FUNCTION_BLOCK FB_InternalPowerSupply implements itf_standardFB

VAR
	IO									: FB_InternalPowerSupply_IO;
	UPS									: FB_UPS;
	InternalPowerDemand					: ST_InternalPowerSupply_PowerDemand;
	b_EMStopActive 						: BOOL := FALSE;
	b_killUPS							: BOOL := FALSE;	
	b_HVDCAllowed						: BOOL;
	
	rtrig_CEEConnected					:	r_trig;
	LowBatShutdownTimer					:	TON;
	
	UPSChargeMode	:	bool;
END_VAR

VAR_IN_OUT CONSTANT
	st_params							: 	ST_InternalPowerSupply_Params;
END_VAR

VAR_INPUT
	st_CoolingDemandSupply				: ST_InternalPowerSupply_PowerDemand;
	st_PowerstackDemandSupply			: ST_InternalPowerSupply_PowerDemand;
	st_ACDCChargerDemandSupply			: ST_InternalPowerSupply_PowerDemand;
	st_DCBusDemandSupply				: ST_InternalPowerSupply_PowerDemand;
	
	b_BusbarACAvailable					: BOOL	:=	FALSE;
	e_BMSPowerstate						: eHVDC_Powerstatus;
	b_ConditioningOnBatteryAllowed		:	BOOL;
END_VAR

VAR_OUTPUT
	Get									: ST_InternalPowerSupply_Get;
	b_HVDC_Enable						: BOOL;
	b_PowerStackACRequired				: BOOL;
END_VAR


var
	b_ACPSU_OK				at %i* :	Bool;
	b_DCPSU_OK				at %i* :	Bool;
	b_CEEInputAvailable		AT %i* : 	Bool;
	b_enableHVDCPSU			AT %Q* :	Bool;
END_VAR

// call functions
UPS(b_24v_available := get.b_24VdcAvailable, st_params := st_params);
	get.UPS REF= UPS.Get;

ACPowerControl(st_params:=st_params, get:=get);
DCPowerControl(st_params:=st_params, b_UPSDemand24VDC := ups.b_UPSDemand24VDC,  get:= get);
HVDCPowerControl(enable := b_HVDCAllowed);

//if ups battery low warning occurs and no 24V is available, charging request failed and the system shuts down.
//If the system is connected to a source (HVDC, CEE, powerlock or internal AC), this is skipped.
//In that case, LowBatteryError will trip a system shutdown
LowBatShutdownTimer(in := UPS.Get.Events.b_BatteryLowWarning AND NOT get.b_24VdcAvailable, PT := st_params.LowBatteryShutdownTimer);
IF LowBatShutdownTimer.Q THEN
	SystemShutdown(TRUE);
END_IF

METHOD PRIVATE ACPowerControl : BOOL
VAR_IN_OUT CONSTANT
	st_params			: ST_Internalpowersupply_params;
END_VAR
VAR_IN_OUT
	get					: ST_InternalPowersupply_get;
END_VAR

VAR_INST
	tof_PowerstackACOffDelay: Tof := (PT := T#10S);
	ton_ACStartupDelay: TON;
	

END_VAR
//if cooling requires 400V, ask powerstack to supply either Main AC or inverter AC.
tof_PowerstackACOffDelay(IN := st_CoolingDemandSupply.b_Demand_400V and b_ConditioningOnBatteryAllowed);
b_PowerStackACRequired := tof_PowerstackACOffDelay.Q;

//after startup delay, internal 400VAC is available
ton_ACStartupDelay(IN := b_BusbarACAvailable, PT:=INT_TO_TIME(st_params.i_ACStartupDelay));
get.b_400VACAvailable := ton_ACstartupDelay.Q;

get.CEEInputActive := b_CEEInputAvailable;
END_METHOD

METHOD DCPowerControl : BOOL
VAR_IN_OUT CONSTANT
	st_params		: ST_Internalpowersupply_params;
	b_UPSDemand24VDC : BOOL;
END_VAR
VAR_IN_OUT
	get				: ST_Internalpowersupply_get;
END_VAR

VAR_INST
	ton_DCPSUStartupDelay: TON;
	ton_ACPSUStartupDelay: TON;
	tof_HVEnableOnUPSBattFailure	:	Tof := (pt := T#10M);
END_VAR
VAR
	DC_Required: BOOL;
END_VAR

ton_DCPSUStartupDelay(IN := get.b_HVDCAvailable, PT:= INT_TO_TIME(st_params.i_DCPSU_StartupDelay));
ton_ACPSUStartupDelay(IN := get.CEEInputActive, PT:= INT_TO_TIME(st_params.i_ACPSU_StartupDelay));

//if psu is not online after the startup delay, raise the fault status.
get.Events.b_ACPSUFault := ton_ACPSUStartupDelay.Q AND NOT b_ACPSU_OK;
get.Events.b_DCPSUFault := ton_DCPSUStartupDelay.Q AND NOT b_DCPSU_OK;

//if CEE psu has no status output, determine based on ups input and CEE AC detection
//	if not UPS.Get.BatteryTestActive then
//		DCPSU_OK := (get.UPS.r_InputVoltage > 20 and get.CEEInputActive);
//	end_if

//if CEE psu has status output, but no ac detection is present. Base AC detection on PSU output.
//get.CEEInputAvailable := DCPSU_OK or main_fast.AcDcCharger.Get.ACDetected;

//if any of the psu's is online, 24V is available
get.b_24VdcAvailable := b_ACPSU_OK OR b_DCPSU_OK;

//if no 400VAC available during 24VDC request, request HVDC ON for LVDC power				
internalPowerDemand.b_Demand_HVDC := NOT get.CEEInputActive AND b_DCPSU_OK;
END_METHOD

METHOD PUBLIC EMstop : BOOL

VAR_INST
	ton_HVDCShutdownTimeout	:	TON := (PT := T#5s);
END_VAR
//return true if done
b_EMStopActive := TRUE;

ton_HVDCShutdownTimeout(in:= get.b_HVDCAvailable);

//if HVDC shutdown takes too long, kill internal HVDC supply to 
get.Events.b_HVDCShutdownTimeExceeded := ton_HVDCShutdownTimeout.Q;

b_HVDCAllowed := FALSE;
//return true when all supplies are lost.
EMStop := NOT(get.b_HVDCAvailable);
END_METHOD

METHOD GetDiagnostics 
VAR_IN_OUT
	AddError		: ARRAY [*] OF FB_AddErrorST;
	a_ActiveEvents	: ARRAY [*] OF ST_ErrorStruct;
	w_Index			: WORD;
END_VAR
//check if this call works:
UPS.GetDiagnostics(AddError := AddError, a_ActiveEvents := a_ActiveEvents, w_Index := w_Index);
 
(*IPS*)
	(*AC PSU fault*)		AddError[w_Index](
			b_ErrorTrig			:= Get.Events.b_ACPSUFault,
			out_ST_Error			:= a_ActiveEvents[w_Index],
			w_ErrorID					:= 1,
			e_objectID				:= eObject_ID.InternalPowerSupply,
			s_Message				:= 'AC PSU fault',
			e_sev					:= eSeverity.Warning,
			t_triggerTime			:= T#3S,
			b_AutoClear			:= TRUE
			);
		w_Index := w_Index +1;
	(*DC PSU fault*)		AddError[w_Index](
			b_ErrorTrig			:= Get.Events.b_DCPSUFault,
			out_ST_Error			:= a_ActiveEvents[w_Index],
			w_ErrorID					:= 2,
			s_Message				:= 'DC PSU fault',
			e_sev					:= eSeverity.Warning,
			t_triggerTime			:= T#3S,
			b_AutoClear			:= TRUE
			);
		w_Index := w_Index +1;
	(*24V fault*)		AddError[w_Index](
			b_ErrorTrig			:= Get.Events.b_DCPSUFault AND Get.Events.b_ACPSUFault,
			out_ST_Error			:= a_ActiveEvents[w_Index],
			w_ErrorID					:= 3,
			s_Message				:= '24V supply failed',
			e_sev					:= eSeverity.QuickShutdown,
			);
		w_Index := w_Index +1;	
// 	(*CEE fuse tripped*)		AddError[w_Index](
// 			b_ErrorTrig			:= Get.Events.b_CEEInputFuseTripped,
// 			out_ST_Error			:= a_ActiveEvents[w_Index],
// 			w_ErrorID					:= 4,
// 			s_Message				:= 'CEE Standby power input fuse error',
// 			e_sev					:= eSeverity.Warning,
// 			b_AutoClear			:= TRUE,
// 			);
// 		w_Index := w_Index +1;
	(*internal grid fuse fault*)		AddError[w_Index](
			b_ErrorTrig		:= Get.Events.b_GridInputFuseTripped,
			out_ST_Error			:= a_ActiveEvents[w_Index],
			w_ErrorID					:= 5,
			s_Message				:= 'Internal supply Grid fuse error',
			e_sev					:= eSeverity.QuickShutdown,
			);
		w_Index := w_Index +1;
		
	(*EMSTOP HVDC shutdown failed*)		AddError[w_Index](
			b_ErrorTrig			:= Get.Events.b_HVDCShutdownTimeExceeded,
			out_ST_Error			:= a_ActiveEvents[w_Index],
			w_ErrorID					:= 6,
			s_Message				:= 'HVDC shutdown sequence failed',
			e_sev					:= eSeverity.QuickShutdown,			//<-- already in emstop, but this is a severe error
			);
		w_Index := w_Index +1;
		
	//Warnings
	(*UPS drained during operation*)		AddError[w_Index](
			b_ErrorTrig				:= UPS.Get.Events.b_BatteryLowWarning,
			out_ST_Error			:= a_ActiveEvents[w_Index],
			w_ErrorID				:= 8,
			s_Message				:= Concat('System shut down in: ', TO_STRING(LowBatShutdownTimer.PT - LowBatShutdownTimer.ET)),
			e_sev					:= eseverity.Warning,
			b_AutoClear				:= TRUE
			);
		w_Index := w_Index +1;
		
	//Warnings
	(*UPS battery low while on battery, initiate shutdown*) 	AddError[w_Index](
			b_ErrorTrig				:= LowBatShutdownTimer.Q,
			out_ST_Error			:= a_ActiveEvents[w_Index],
			w_ErrorID				:= 9,
			s_Message				:= 'Shutdown initiated: Halt system operation',
			e_sev					:= eseverity.QuickShutdown,
			b_AutoClear				:= TRUE
			);
		w_Index := w_Index +1;
END_METHOD

METHOD GetWearCounters : BOOL
VAR_INST
	ACPsuPoH				:	FB_Varlogger;
	DCPsuPoh				:	FB_Varlogger;
END_VAR

ACPsuPoH(				TriggerInput := IO.ACPSU_OK, 
						LogItemGroup :=  eLogItemGroupID.InternalPowerSupply, 
						LogItemName := 'AcPsuHrs', 
						LogType := eLogTypes.TrackOnTime);

DCPsuPoh(				TriggerInput := io.DCPSU_OK, 
						LogItemGroup :=  eLogItemGroupID.InternalPowerSupply, 
						LogItemName := 'DcPsuHrs', 
						LogType := eLogTypes.TrackOnTime);	

UPS.getWearCounters();
END_METHOD

METHOD HVDC_disable : BOOL;
b_HVDCAllowed := FALSE;
HVDC_disable := NOT b_HVDC_Enable;
END_METHOD

METHOD HVDC_Enable : BOOL
VAR_INPUT
END_VAR
b_HVDCAllowed := True;
END_METHOD

METHOD PRIVATE HVDCPowerControl : BOOL

VAR_INPUT
	enable		: BOOL;
END_VAR

VAR_INST
	TON_HVONDelay : TON := (PT := T#1S);
	TOF_HVOnDelay : TOF := (PT := T#1S);
END_VAR
//The powerstack demands HVDC directly. 
TOF_HVOnDelay(in:=	st_powerstackdemandsupply.b_Demand_HVDC OR 
					InternalPowerDemand.b_Demand_HVDC or 
					st_DCBusDemandSupply.b_Demand_HVDC or 
					st_ACDCChargerDemandSupply.b_Demand_HVDC or
					st_CoolingDemandSupply.b_Demand_HVDC);
b_HVDC_Enable := TOF_HVOnDelay.Q AND NOT b_EMStopActive AND enable;


TON_HVONDelay(in:= e_BMSPowerstate = eHVDC_Powerstatus.ON);
IF TON_HVONDelay.Q THEN
	IO.b_DCPsuEnable := TRUE;
	get.b_HVDCAvailable := TRUE;
ELSE
	IO.b_DCPsuEnable := FALSE;
	get.b_HVDCAvailable := FALSE;
END_IF
END_METHOD

{warning 'Add method implementation '}
METHOD Init : BOOL
END_METHOD

METHOD Reset : BOOL
//reset system
b_EMStopActive := FALSE;
get.Events.b_HVDCShutdownTimeExceeded := FALSE;
b_HVDCAllowed := TRUE;

Reset := NOT get.Events.b_GridInputFuseTripped;
//return true if ok
END_METHOD

METHOD SystemShutdown : BOOL

VAR_INPUT
	TimedShutdown		:	BOOL;
END_VAR

IF NOT TimedShutdown THEN
	get.Events.b_CEEPreventsShutdown := b_CEEInputAvailable;
	b_enableHVDCPSU	:= false;
	UPS.Shutdown();
END_IF
END_METHOD

END_FUNCTION_BLOCK

(* stored: Version 1.1.0.1, ProductVersion 3.1.4026.18
   POU FB_InternalPowerSupply: Id {99b5595d-91f9-4503-8fb7-aed8af10f6d8}, SpecialFunc None
   Folder Private: Id {09cc00c9-9aef-44dd-8920-4fac26adde0c}
   Method ACPowerControl: Id {5916b7c6-c369-43a6-ad0f-f820d571c778}
   Method DCPowerControl: Id {4cfaa935-ee98-4c42-8d5b-fbc6199322b8}
   Method EMstop: Id {4866248a-59ca-4029-a026-7364cef193b4}
   Method GetDiagnostics: Id {f562ae03-1873-4d82-904d-4e0cc41d7903}
   Method GetWearCounters: Id {031c6c2d-7de1-4023-a28b-11b52efeabe4}
   Method HVDC_disable: Id {7ef0694f-e03e-47bc-9226-19e673c0f031}
   Method HVDC_Enable: Id {eb5577ab-d3e1-4e62-a922-b65df6a78269}
   Method HVDCPowerControl: Id {ed7ee3c2-5980-4244-9ba9-7c622b5d790a}
   Method Init: Id {49b9e4e0-90d3-412a-b77c-7ecb0b10dedf}
   Method Reset: Id {d1725ace-f077-4c1f-9e1a-d4d8e986182f}
   Method SystemShutdown: Id {665b7361-b80d-4473-8f04-c6493ebb91db} *)
